// TIA Portal V16 export
// export: Created 2023-03-29T11:04:36.6836641Z, ExportSetting WithDefaults, DisplayName Totally Integrated Automation Portal, DisplayVersion V16 Update 6, DisplayName TIA Portal Version Control Interface, DisplayVersion V16 Update 2, DisplayName TIA Portal Openness, DisplayVersion V16 Update 6, DisplayName STEP 7 Professional, DisplayVersion V16 Update 6, DisplayName STEP 7 Safety, DisplayVersion V16, DisplayName WinCC Advanced, DisplayVersion V16 Update 6
FUNCTION_BLOCK "Modbus_TCP"   // FB6, LAD
TITLE = Wywołanie funkcji MB_Server
{ S7_Optimized_Access := 'TRUE' }
AUTHOR : rtecmer
VERSION : 0.1
// stored: AutoNumber true, IsIECCheckEnabled false, IsRetainMemResEnabled false, MemoryReserve 100, SetENOAutomatically false, UDAEnableTagReadback false
   VAR_TEMP   // added for the SCL form of the ladder/FBD networks
      _w1 : Bool;
   END_VAR
BEGIN

REGION Network 1: Sewrer
   // Wpisywane z PLC 2 Zbiorniki
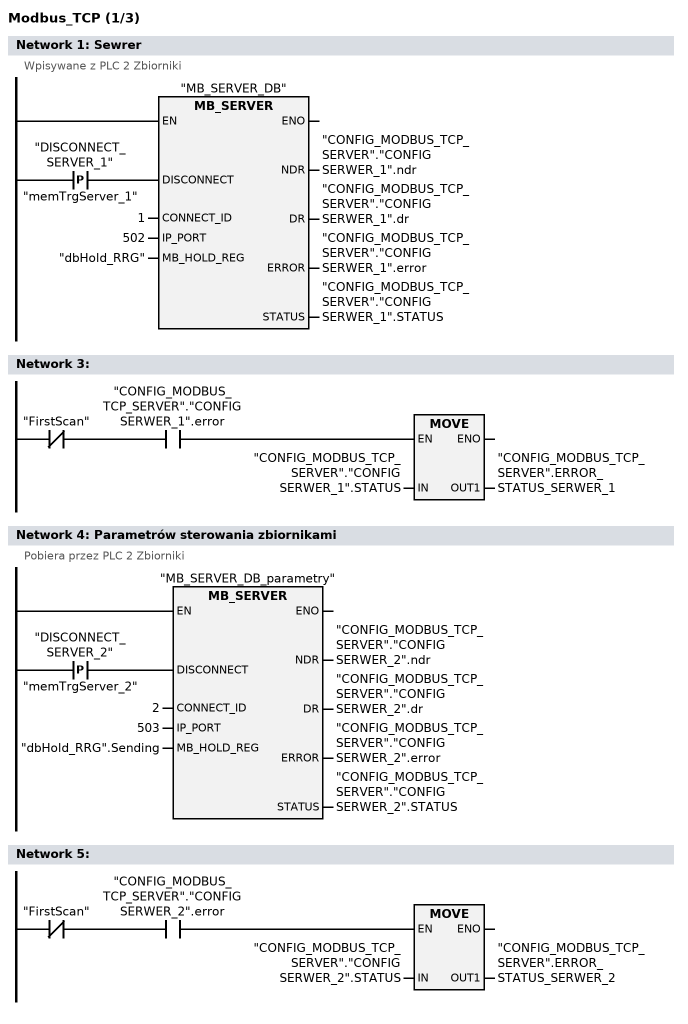
   RUNG wire#powerrail
      { S7_Templates := "[card1200 := 1, card1500 := 0]" } "MB_SERVER_DB".MB_SERVER(DISCONNECT := wire#w1, CONNECT_ID := 1, IP_PORT := 502, MB_HOLD_REG := "dbHold_RRG", NDR => "CONFIG_MODBUS_TCP_SERVER"."CONFIG SERWER_1".ndr, DR => "CONFIG_MODBUS_TCP_SERVER"."CONFIG SERWER_1".dr, ERROR => "CONFIG_MODBUS_TCP_SERVER"."CONFIG SERWER_1".error, STATUS => "CONFIG_MODBUS_TCP_SERVER"."CONFIG SERWER_1".STATUS)
   END_RUNG
   RUNG wire#powerrail
      P_Contact(operand := "DISCONNECT_SERVER_1", bit := "memTrgServer_1")
   END_RUNG wire#w1
   // the same network as SCL:
   #_w1 := "DISCONNECT_SERVER_1" AND NOT "memTrgServer_1";   // rising edge of "DISCONNECT_SERVER_1"
   "memTrgServer_1" := "DISCONNECT_SERVER_1";
   "MB_SERVER_DB"(DISCONNECT := #_w1,   // MB_SERVER
                  CONNECT_ID := 1,
                  IP_PORT := 502,
                  MB_HOLD_REG := "dbHold_RRG",
                  NDR => "CONFIG_MODBUS_TCP_SERVER"."CONFIG SERWER_1".ndr,
                  DR => "CONFIG_MODBUS_TCP_SERVER"."CONFIG SERWER_1".dr,
                  ERROR => "CONFIG_MODBUS_TCP_SERVER"."CONFIG SERWER_1".error,
                  STATUS => "CONFIG_MODBUS_TCP_SERVER"."CONFIG SERWER_1".STATUS);
END_REGION

REGION Network 3
   RUNG wire#powerrail
      I_Contact( "FirstScan" )
      Contact( "CONFIG_MODBUS_TCP_SERVER"."CONFIG SERWER_1".error )
      Move(in := "CONFIG_MODBUS_TCP_SERVER"."CONFIG SERWER_1".STATUS, out1 => "CONFIG_MODBUS_TCP_SERVER".ERROR_STATUS_SERWER_1)
   END_RUNG
   // the same network as SCL:
   IF NOT "FirstScan" AND "CONFIG_MODBUS_TCP_SERVER"."CONFIG SERWER_1".error THEN
       "CONFIG_MODBUS_TCP_SERVER".ERROR_STATUS_SERWER_1 := "CONFIG_MODBUS_TCP_SERVER"."CONFIG SERWER_1".STATUS;
   END_IF;
END_REGION

REGION Network 4: Parametrów sterowania zbiornikami
   // Pobiera przez PLC 2 Zbiorniki
   RUNG wire#powerrail
      { S7_Templates := "[card1200 := 1, card1500 := 0]" } "MB_SERVER_DB_parametry".MB_SERVER(DISCONNECT := wire#w1, CONNECT_ID := 2, IP_PORT := 503, MB_HOLD_REG := "dbHold_RRG".Sending, NDR => "CONFIG_MODBUS_TCP_SERVER"."CONFIG SERWER_2".ndr, DR => "CONFIG_MODBUS_TCP_SERVER"."CONFIG SERWER_2".dr, ERROR => "CONFIG_MODBUS_TCP_SERVER"."CONFIG SERWER_2".error, STATUS => "CONFIG_MODBUS_TCP_SERVER"."CONFIG SERWER_2".STATUS)
   END_RUNG
   RUNG wire#powerrail
      P_Contact(operand := "DISCONNECT_SERVER_2", bit := "memTrgServer_2")
   END_RUNG wire#w1
   // the same network as SCL:
   #_w1 := "DISCONNECT_SERVER_2" AND NOT "memTrgServer_2";   // rising edge of "DISCONNECT_SERVER_2"
   "memTrgServer_2" := "DISCONNECT_SERVER_2";
   "MB_SERVER_DB_parametry"(DISCONNECT := #_w1,   // MB_SERVER
                           CONNECT_ID := 2,
                           IP_PORT := 503,
                           MB_HOLD_REG := "dbHold_RRG".Sending,
                           NDR => "CONFIG_MODBUS_TCP_SERVER"."CONFIG SERWER_2".ndr,
                           DR => "CONFIG_MODBUS_TCP_SERVER"."CONFIG SERWER_2".dr,
                           ERROR => "CONFIG_MODBUS_TCP_SERVER"."CONFIG SERWER_2".error,
                           STATUS => "CONFIG_MODBUS_TCP_SERVER"."CONFIG SERWER_2".STATUS);
END_REGION

REGION Network 5
   RUNG wire#powerrail
      I_Contact( "FirstScan" )
      Contact( "CONFIG_MODBUS_TCP_SERVER"."CONFIG SERWER_2".error )
      Move(in := "CONFIG_MODBUS_TCP_SERVER"."CONFIG SERWER_2".STATUS, out1 => "CONFIG_MODBUS_TCP_SERVER".ERROR_STATUS_SERWER_2)
   END_RUNG
   // the same network as SCL:
   IF NOT "FirstScan" AND "CONFIG_MODBUS_TCP_SERVER"."CONFIG SERWER_2".error THEN
       "CONFIG_MODBUS_TCP_SERVER".ERROR_STATUS_SERWER_2 := "CONFIG_MODBUS_TCP_SERVER"."CONFIG SERWER_2".STATUS;
   END_IF;
END_REGION

REGION Network 6: Czasy zadawane
   // Pobiera PLC 2 Zbiorniki
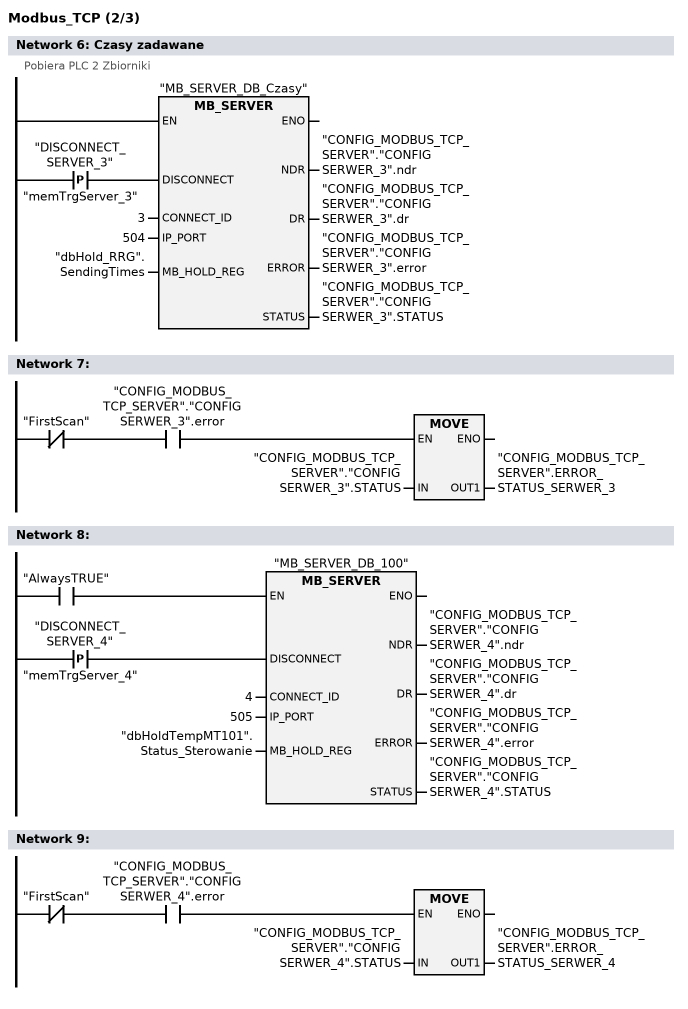
   RUNG wire#powerrail
      { S7_Templates := "[card1200 := 1, card1500 := 0]" } "MB_SERVER_DB_Czasy".MB_SERVER(DISCONNECT := wire#w1, CONNECT_ID := 3, IP_PORT := 504, MB_HOLD_REG := "dbHold_RRG".SendingTimes, NDR => "CONFIG_MODBUS_TCP_SERVER"."CONFIG SERWER_3".ndr, DR => "CONFIG_MODBUS_TCP_SERVER"."CONFIG SERWER_3".dr, ERROR => "CONFIG_MODBUS_TCP_SERVER"."CONFIG SERWER_3".error, STATUS => "CONFIG_MODBUS_TCP_SERVER"."CONFIG SERWER_3".STATUS)
   END_RUNG
   RUNG wire#powerrail
      P_Contact(operand := "DISCONNECT_SERVER_3", bit := "memTrgServer_3")
   END_RUNG wire#w1
   // the same network as SCL:
   #_w1 := "DISCONNECT_SERVER_3" AND NOT "memTrgServer_3";   // rising edge of "DISCONNECT_SERVER_3"
   "memTrgServer_3" := "DISCONNECT_SERVER_3";
   "MB_SERVER_DB_Czasy"(DISCONNECT := #_w1,   // MB_SERVER
                        CONNECT_ID := 3,
                        IP_PORT := 504,
                        MB_HOLD_REG := "dbHold_RRG".SendingTimes,
                        NDR => "CONFIG_MODBUS_TCP_SERVER"."CONFIG SERWER_3".ndr,
                        DR => "CONFIG_MODBUS_TCP_SERVER"."CONFIG SERWER_3".dr,
                        ERROR => "CONFIG_MODBUS_TCP_SERVER"."CONFIG SERWER_3".error,
                        STATUS => "CONFIG_MODBUS_TCP_SERVER"."CONFIG SERWER_3".STATUS);
END_REGION

REGION Network 7
   RUNG wire#powerrail
      I_Contact( "FirstScan" )
      Contact( "CONFIG_MODBUS_TCP_SERVER"."CONFIG SERWER_3".error )
      Move(in := "CONFIG_MODBUS_TCP_SERVER"."CONFIG SERWER_3".STATUS, out1 => "CONFIG_MODBUS_TCP_SERVER".ERROR_STATUS_SERWER_3)
   END_RUNG
   // the same network as SCL:
   IF NOT "FirstScan" AND "CONFIG_MODBUS_TCP_SERVER"."CONFIG SERWER_3".error THEN
       "CONFIG_MODBUS_TCP_SERVER".ERROR_STATUS_SERWER_3 := "CONFIG_MODBUS_TCP_SERVER"."CONFIG SERWER_3".STATUS;
   END_IF;
END_REGION

REGION Network 8
   RUNG wire#powerrail
      Contact( "AlwaysTRUE" )
      { S7_Templates := "[card1200 := 1, card1500 := 0]" } "MB_SERVER_DB_100".MB_SERVER(DISCONNECT := wire#w1, CONNECT_ID := 4, IP_PORT := 505, MB_HOLD_REG := "dbHoldTempMT101".Status_Sterowanie, NDR => "CONFIG_MODBUS_TCP_SERVER"."CONFIG SERWER_4".ndr, DR => "CONFIG_MODBUS_TCP_SERVER"."CONFIG SERWER_4".dr, ERROR => "CONFIG_MODBUS_TCP_SERVER"."CONFIG SERWER_4".error, STATUS => "CONFIG_MODBUS_TCP_SERVER"."CONFIG SERWER_4".STATUS)
   END_RUNG
   RUNG wire#powerrail
      P_Contact(operand := "DISCONNECT_SERVER_4", bit := "memTrgServer_4")
   END_RUNG wire#w1
   // the same network as SCL:
   #_w1 := "DISCONNECT_SERVER_4" AND NOT "memTrgServer_4";   // rising edge of "DISCONNECT_SERVER_4"
   "memTrgServer_4" := "DISCONNECT_SERVER_4";
   IF "AlwaysTRUE" THEN
       "MB_SERVER_DB_100"(DISCONNECT := #_w1,   // MB_SERVER
                          CONNECT_ID := 4,
                          IP_PORT := 505,
                          MB_HOLD_REG := "dbHoldTempMT101".Status_Sterowanie,
                          NDR => "CONFIG_MODBUS_TCP_SERVER"."CONFIG SERWER_4".ndr,
                          DR => "CONFIG_MODBUS_TCP_SERVER"."CONFIG SERWER_4".dr,
                          ERROR => "CONFIG_MODBUS_TCP_SERVER"."CONFIG SERWER_4".error,
                          STATUS => "CONFIG_MODBUS_TCP_SERVER"."CONFIG SERWER_4".STATUS);
   END_IF;
END_REGION

REGION Network 9
   RUNG wire#powerrail
      I_Contact( "FirstScan" )
      Contact( "CONFIG_MODBUS_TCP_SERVER"."CONFIG SERWER_4".error )
      Move(in := "CONFIG_MODBUS_TCP_SERVER"."CONFIG SERWER_4".STATUS, out1 => "CONFIG_MODBUS_TCP_SERVER".ERROR_STATUS_SERWER_4)
   END_RUNG
   // the same network as SCL:
   IF NOT "FirstScan" AND "CONFIG_MODBUS_TCP_SERVER"."CONFIG SERWER_4".error THEN
       "CONFIG_MODBUS_TCP_SERVER".ERROR_STATUS_SERWER_4 := "CONFIG_MODBUS_TCP_SERVER"."CONFIG SERWER_4".STATUS;
   END_IF;
END_REGION

REGION Network 10: Reakcja na błąd komunikacji
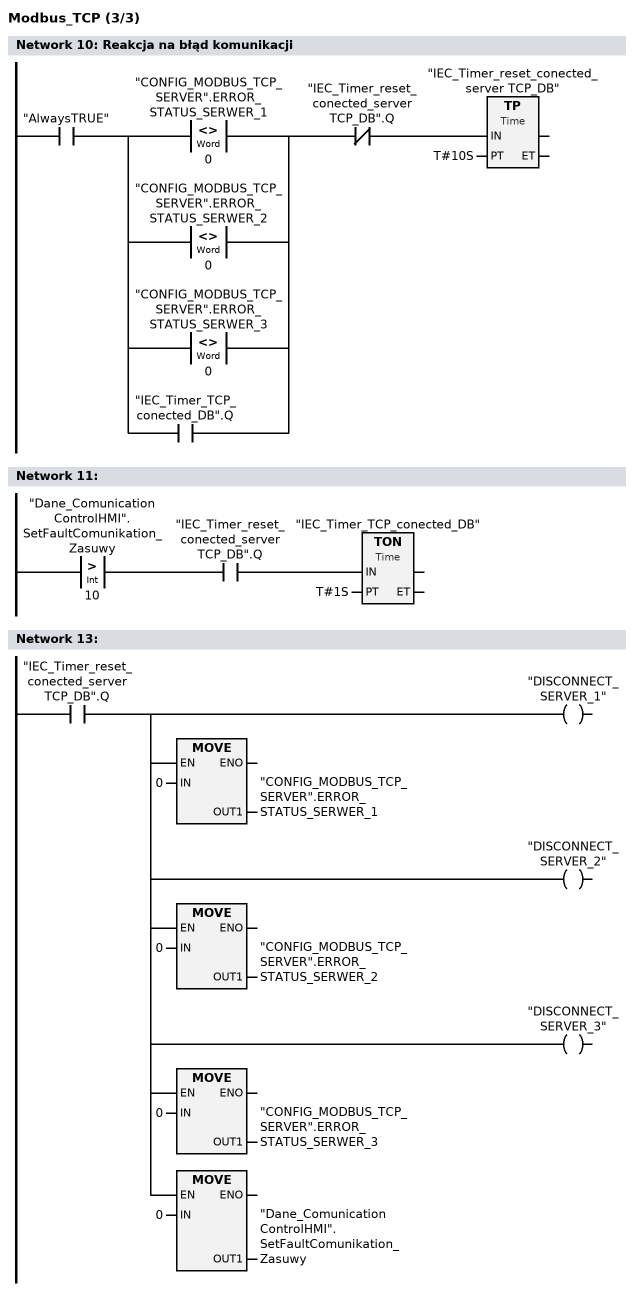
   RUNG wire#powerrail
      Contact( "AlwaysTRUE" )
      wire#w1
      { S7_Templates := "SrcType := Word" } NE_Contact(in1 := "CONFIG_MODBUS_TCP_SERVER".ERROR_STATUS_SERWER_1, in2 := 0)
      wire#w2
      I_Contact( "IEC_Timer_reset_conected_server TCP_DB".Q )
      { S7_Templates := "time_type := Time" } "IEC_Timer_reset_conected_server TCP_DB".TP(pt := T#10S, et =>)
   END_RUNG
   RUNG wire#w1
      { S7_Templates := "SrcType := Word" } NE_Contact(in1 := "CONFIG_MODBUS_TCP_SERVER".ERROR_STATUS_SERWER_2, in2 := 0)
   END_RUNG wire#w2
   RUNG wire#w1
      { S7_Templates := "SrcType := Word" } NE_Contact(in1 := "CONFIG_MODBUS_TCP_SERVER".ERROR_STATUS_SERWER_3, in2 := 0)
   END_RUNG wire#w2
   RUNG wire#w1
      Contact( "IEC_Timer_TCP_conected_DB".Q )
   END_RUNG wire#w2
   // the same network as SCL:
   "IEC_Timer_reset_conected_server TCP_DB".TP(IN := "AlwaysTRUE" AND (("CONFIG_MODBUS_TCP_SERVER".ERROR_STATUS_SERWER_1 <> 0) OR ("CONFIG_MODBUS_TCP_SERVER".ERROR_STATUS_SERWER_2 <> 0) OR ("CONFIG_MODBUS_TCP_SERVER".ERROR_STATUS_SERWER_3 <> 0) OR "IEC_Timer_TCP_conected_DB".Q) AND NOT "IEC_Timer_reset_conected_server TCP_DB".Q,
                           PT := T#10S);
END_REGION

REGION Network 11
   RUNG wire#powerrail
      { S7_Templates := "SrcType := Int" } GT_Contact(in1 := "Dane_ComunicationControlHMI".SetFaultComunikation_Zasuwy, in2 := 10)
      Contact( "IEC_Timer_reset_conected_server TCP_DB".Q )
      { S7_Templates := "time_type := Time" } "IEC_Timer_TCP_conected_DB".TON(pt := T#1S, et =>)
   END_RUNG
   // the same network as SCL:
   "IEC_Timer_TCP_conected_DB".TON(IN := ("Dane_ComunicationControlHMI".SetFaultComunikation_Zasuwy > 10) AND "IEC_Timer_reset_conected_server TCP_DB".Q,
                           PT := T#1S);
END_REGION

REGION Network 13
   RUNG wire#powerrail
      Contact( "IEC_Timer_reset_conected_server TCP_DB".Q )
      wire#w1
      Coil( "DISCONNECT_SERVER_1" )
   END_RUNG
   RUNG wire#w1
      Move(in := 0, out1 => "CONFIG_MODBUS_TCP_SERVER".ERROR_STATUS_SERWER_1)
   END_RUNG
   RUNG wire#w1
      Coil( "DISCONNECT_SERVER_2" )
   END_RUNG
   RUNG wire#w1
      Move(in := 0, out1 => "CONFIG_MODBUS_TCP_SERVER".ERROR_STATUS_SERWER_2)
   END_RUNG
   RUNG wire#w1
      Coil( "DISCONNECT_SERVER_3" )
   END_RUNG
   RUNG wire#w1
      Move(in := 0, out1 => "CONFIG_MODBUS_TCP_SERVER".ERROR_STATUS_SERWER_3)
   END_RUNG
   RUNG wire#w1
      Move(in := 0, out1 => "Dane_ComunicationControlHMI".SetFaultComunikation_Zasuwy)
   END_RUNG
   // the same network as SCL:
   "DISCONNECT_SERVER_1" := "IEC_Timer_reset_conected_server TCP_DB".Q;
   IF "IEC_Timer_reset_conected_server TCP_DB".Q THEN
       "CONFIG_MODBUS_TCP_SERVER".ERROR_STATUS_SERWER_1 := 0;
   END_IF;
   "DISCONNECT_SERVER_2" := "IEC_Timer_reset_conected_server TCP_DB".Q;
   IF "IEC_Timer_reset_conected_server TCP_DB".Q THEN
       "CONFIG_MODBUS_TCP_SERVER".ERROR_STATUS_SERWER_2 := 0;
   END_IF;
   "DISCONNECT_SERVER_3" := "IEC_Timer_reset_conected_server TCP_DB".Q;
   IF "IEC_Timer_reset_conected_server TCP_DB".Q THEN
       "CONFIG_MODBUS_TCP_SERVER".ERROR_STATUS_SERWER_3 := 0;
       "Dane_ComunicationControlHMI".SetFaultComunikation_Zasuwy := 0;
   END_IF;
END_REGION
END_FUNCTION_BLOCK
